{attribute 'GeneratedUsingTerminal: EP6090-0000-0017'}
{attribute addProperty BoxType "EP6090-0000-0017"}
{attribute addProperty Id "Value_rowAT %Q*ARRAY[0..1] OF INT4"}
{attribute addProperty CRC "4003442326"}
{attribute addProperty Size "4"}
TYPE DIS_Outputs_6C9BFFEE :
STRUCT
	{attribute addProperty Name "Value_row"}
	Value_row AT %Q* : ARRAY[0..1] OF INT;
END_STRUCT
END_TYPE

(* stored: Version 1.2.0.0, ProductVersion 3.1.4024.9
   DUT DIS_Outputs_6C9BFFEE: Id {1c9caf8c-4ebf-41cd-b946-9dc5d8f2b428} *)
